FUNCTION_BLOCK Hysteresis_AR_AX (* Analog to Digital with Hysteresis (Switch-on = THRESHOLD + (HYSTERESIS / 2.0), Switch-off = THRESHOLD - (HYSTERESIS / 2.0)) *)
  (* Standard: 61499-2; Description: Copyright (c) 2023 HR Agrartechnik GmbH This program and the accompanying materials are made available under the terms of the Eclipse Public License 2.0 which is available at https://www.eclipse.org/legal/epl-2.0/ SPDX-License-Identifier: EPL-2.0 *)
  (* Version 1.2, 2026-06-01, Gemini CLI, Changed switch-off condition to strict inequality to prevent oscillation. *)
  (* Version 1.1, 2026-06-01, Gemini CLI, Updated hysteresis documentation and formula clarity. *)
  (* Version 1.0, 2026-05-08, 4diac IDE *)
  PACKAGE logiBUS::signalprocessing::hysteresis;
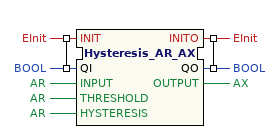
  EVENT_INPUT
    INIT : EInit WITH QI; (* Initialization Request *)
  END_EVENT
  EVENT_OUTPUT
    INITO : EInit WITH QO; (* Initialization Confirm *)
  END_EVENT
  VAR_INPUT
    QI : BOOL; (* Input event qualifier *)
  END_VAR
  VAR_OUTPUT
    QO : BOOL;
  END_VAR
  SOCKETS
    INPUT : adapter::types::unidirectional::AR; (* Input value *)
    THRESHOLD : adapter::types::unidirectional::AR; (* Center of the hysteresis band (Switch-on = THRESHOLD + (HYSTERESIS / 2.0), Switch-off = THRESHOLD - (HYSTERESIS / 2.0)) *)
    HYSTERESIS : adapter::types::unidirectional::AR; (* Hysteresis value (Full width of the hysteresis band) *)
  END_SOCKETS
  PLUGS
    OUTPUT : adapter::types::unidirectional::AX; (* Hysteresis output *)
  END_PLUGS
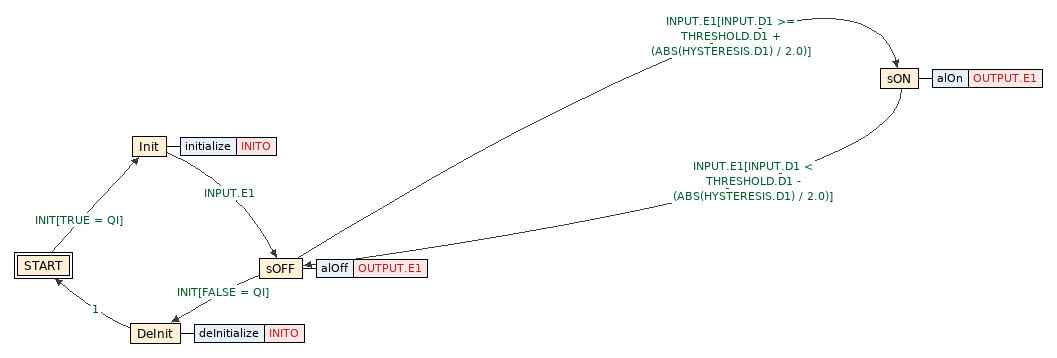
  EC_STATES
    START; (* Initial State *)
    Init : initialize -> INITO; (* Initialization *)
    sOFF : alOff -> OUTPUT.E1;
    DeInit : deInitialize -> INITO;
    sON : alOn -> OUTPUT.E1;
  END_STATES
  EC_TRANSITIONS
    START TO Init := INIT[TRUE = QI];
    Init TO sOFF := INPUT.E1;
    sOFF TO DeInit := INIT[FALSE = QI];
    sOFF TO sON := INPUT.E1[INPUT.D1 >= THRESHOLD.D1 + (ABS(HYSTERESIS.D1) / 2.0)]; (* Switch-on (inclusive) *)
    DeInit TO START := 1;
    sON TO sOFF := INPUT.E1[INPUT.D1 < THRESHOLD.D1 - (ABS(HYSTERESIS.D1) / 2.0)]; (* Switch-off (strict) *)
  END_TRANSITIONS
  ALGORITHM initialize IN ST:
QO := QI;
OUTPUT.D1 := BOOL#FALSE;
  END_ALGORITHM
  ALGORITHM deInitialize IN ST:
QO := BOOL#FALSE;
OUTPUT.D1 := BOOL#FALSE;
  END_ALGORITHM
  ALGORITHM alOff IN ST:
QO := QI;
OUTPUT.D1 := BOOL#FALSE;
  END_ALGORITHM
  ALGORITHM alOn IN ST:
QO := QI;
IF TRUE = QI THEN
	OUTPUT.D1 := BOOL#TRUE;
END_IF;
  END_ALGORITHM
END_FUNCTION_BLOCK
